TYPE ST_AirPressureOutCmd :
STRUCT
    Reserved : BOOL; // passive monitor: no command result
END_STRUCT
END_TYPE

(* stored: Version 1.1.0.1, ProductVersion 3.1.4024.12
   DUT ST_AirPressureOutCmd: Id {ee63f085-2b36-4754-a552-c9d99ec4e431} *)
